PROGRAM PositionHorAxis
VAR
END_VAR

HAVL.axis.ReadStatus();

HAVL.axisPower(
	Axis:= HAVL.axis,
	Enable:= HAVL.enable,
	Enable_Positive:= HAVL.enable,
	Enable_Negative:= HAVL.enable,
	Override:= HAVL.override,
	BufferMode:= ,
	Options:= ,
	Status=> HAVL.running,
	Busy=> ,
	Active=> ,
	Error=> ,
	ErrorID=> HAVL.currentError
);

HAVL.axisMoveAbsolute(
	Axis:= HAVL.axis,
	Execute:= HAVL.enableMove,
	Position:= HAVL.targetPosition,
	Velocity:= HAVL.targetVelocity,
	Acceleration:= ,
	Deceleration:= ,
	Jerk:= ,
	BufferMode:= ,
	Options:= ,
	Done=> HAVL.done,
	Busy=> HAVL.busy,
	Active=> ,
	CommandAborted=> ,
	Error=> ,
	ErrorID=> HAVL.currentError 
);

IF HAVL.busy THEN
	HAVL.axisReadActualPosition(Axis := HAVL.axis, Enable := TRUE, Valid=>, Busy=>, Error=>, ErrorID=>, Position=> HAVL.actualPosition);
END_IF
HAVL.actualPositionInt := LREAL_TO_INT(HAVL.actualPosition);

HAVL.axisErrorReset(Axis := HAVL.axis, Execute := HAVL.resetError, Done =>, Error =>, ErrorID => HAVL.currentError);

END_PROGRAM

(* stored: Version 1.1.0.1, ProductVersion 3.1.4024.6
   POU PositionHorAxis: Id {83c65318-1354-4401-acbf-74659e54a225}, SpecialFunc None *)
